TYPE ST_LoadingBottleParams :
STRUCT
	rLoadingDetectionFrom :REAL;
	rLoadingDetectionTo	:REAL;
END_STRUCT
END_TYPE

(* stored: Version 1.1.0.1, ProductVersion 3.1.4024.15
   DUT ST_LoadingBottleParams: Id {0d2addef-ee45-4ee7-91aa-ebf3db41cfd0} *)
